(* IEC 61131-3 sources: PL-ultimate-llm/languages/IEC 61131-3/programs/7b6837673cfd482fb10d9964ab982a9f65dad7a4403564719202f03dd3985a00, 1 file *)

(* ---- code.st ---- *)
PROGRAM FibonacciCalc
VAR
    n      : INT := 10;
    a, b   : INT;
    temp   : INT;
    i      : INT;
    result : INT;
END_VAR

(* Compute the nth Fibonacci number using iteration *)
a := 0;
b := 1;
FOR i := 1 TO n DO
    temp := a + b;
    a := b;
    b := temp;
END_FOR;
result := a;
END_PROGRAM
